Fanuc KAREL source: kt00488.KL

PROGRAM KT00488
%STACKSIZE=65535
%PRIORITY=65535
%NOLOCKGROUP
VAR
P1 : POSITION
P2 : JOINTPOS9
OUT : BOOLEAN
BEGIN
-- UNRESOLVED_PC line 8 opcodes [49 49 7E AC 23] marker_code=0
END KT00488
